FUNCTION F_Variable_FromUI_Interlock: BOOL

END_FUNCTION

(* stored: Version 1.1.0.1, ProductVersion 3.1.4024.15
   POU F_Variable_FromUI_Interlock: Id {24dd70c4-f47e-49a1-9f71-9d56635c4d74}, SpecialFunc None *)
